INTERFACE IActuator

METHOD Cycle : BOOL
VAR_INPUT
END_VAR
END_METHOD

METHOD Extend : BOOL
VAR_INPUT
END_VAR
END_METHOD

PROPERTY Extended : BOOL
GET
END_GET
END_PROPERTY

METHOD Retract : BOOL
VAR_INPUT
END_VAR
END_METHOD

PROPERTY Retracted : BOOL
GET
END_GET
END_PROPERTY

END_INTERFACE

(* stored: Version 1.1.0.1, ProductVersion 3.1.4024.12
   Itf IActuator: Id {a3ab8863-4a3e-4efe-8fe3-613317ef6a74}
   Method Cycle: Id {142252cc-d944-464a-81a3-9aa66de2f56f}
   Method Extend: Id {2ff4ea27-8d78-4e8d-841c-8dde8ed66a43}
   Property Extended: Id {559518b5-c18a-4148-93c4-bf502c2fe720}
   Get Get: Id {8d559355-eb15-463b-83b9-25e6e8daf3ac}
   Method Retract: Id {92118b42-44eb-415d-9973-473424eac790}
   Property Retracted: Id {0f8722ee-99b4-4388-8341-ad7e7516b2ab}
   Get Get: Id {634e679d-19e2-47bf-98d0-96b878f945be} *)
